// TIA Portal V20 export
DATA_BLOCK "DB_VisuColor"   // DB2
// stored: Access Published, MemoryReserve 100, Namespace Global
   VAR
      Line : Struct
         ProductionLine : Struct
            GlobalStatus : Int;
            Conveyor : Array[_.gminProductionLine.._.gmaxProductionLine] of Int;
         END_STRUCT;
         EmptyLine : Struct
            GlobalStatus : Int;
            Conveyor : Array[_.gminEmptyLine.._.gmaxEmptyLine] of Int;
         END_STRUCT;
         PackedLine : Struct
            GlobalStatus : Int;
            Conveyor : Array[_.gminPackedLine.._.gmaxPackedLine] of Int;
         END_STRUCT;
      END_STRUCT;
   END_VAR
BEGIN
END_DATA_BLOCK
